// TwinCAT 3 PLC project PLC
// ProgramVersion: 3.1.4024.0
// libraries:
//   Tc2_Standard, * (Beckhoff Automation GmbH)
//   Tc2_System, * (Beckhoff Automation GmbH)
//   Tc3_Module, * (Beckhoff Automation GmbH)
// project tree:
//   / GlobalTextList.TcGTLO, PlcTask.TcTTO, Visualization Manager.TcVMO (not stored), Visualization.TcVIS
//   POUs/ MAIN.TcPOU
// real-time tasks:
//   TASK PlcTask: cycle T#10ms, priority 20, ADS port 350

CONFIGURATION PLC
    RESOURCE PLC ON TwinCAT3
        TASK PlcTask(INTERVAL := T#10ms, PRIORITY := 20);
        PROGRAM MAIN WITH PlcTask : MAIN;
    END_RESOURCE
END_CONFIGURATION

// ---- POUs/MAIN.TcPOU
PROGRAM MAIN
VAR
	StartPb					:	BOOL;
	StopPB					:	BOOL;
	MotorStart				: 	RS;
	Motor					: 	BOOL;
	ProductCnt				: 	CTU;
	LightBarrierSensor		: 	BOOL;
	ProductCounter			: 	WORD;
	TrayChange				: 	BOOL;
END_VAR
VAR // added by the converter: edge detectors and wires of the graphical bodies
    _w1 : ANY;
END_VAR

MotorStart(SET := StartPb, RESET1 := StopPB); // RS
ProductCnt(CU := Motor AND LightBarrierSensor, RESET := _w1, PV := 5); // CTU
ProductCounter := ProductCnt.CV;
Motor := MotorStart.Q1 AND NOT ProductCnt.Q;
_w1 := TrayChange AND ProductCnt.Q;

END_PROGRAM

// ---- GlobalTextList.TcGTLO
TEXTLIST GlobalTextList
  899 = '%s'
  542 = 'Change Tray'
  722 = 'Light Barrier'
  329 = 'Motor'
  959 = 'Please Change the Tray'
  663 = 'Product amount: \n%s'
  828 = 'Product amount: %s'
  814 = 'RUN'
  239 = 'START'
  872 = 'STOP'
END_TEXTLIST

// ---- Visualization.TcVIS
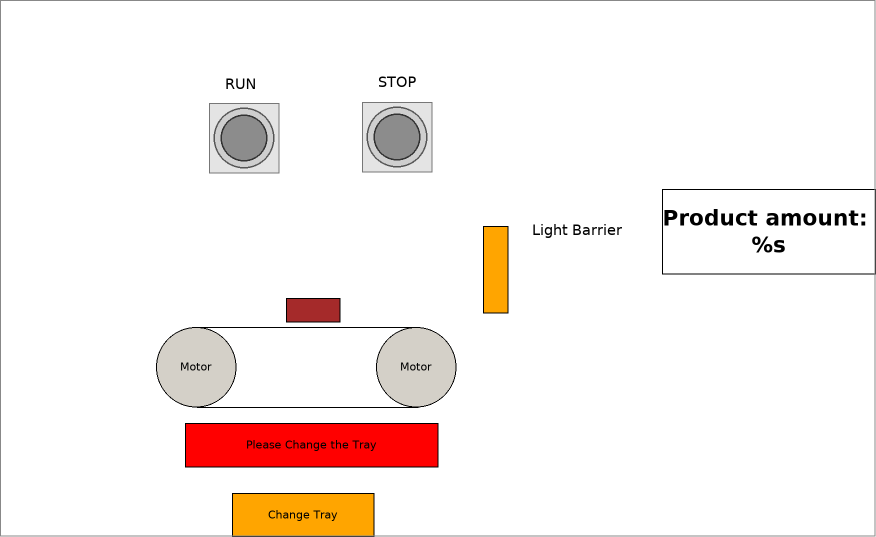
VISUALIZATION Visualization  // 876x537
    PushSwitchLed (209,103 70x70), variable: MAIN.StartPb, behaviour: TAP, style: Switch-PushSwitchLed-Gray
    PushSwitchLed (362,102 70x70), variable: MAIN.StopPB, behaviour: TAP, style: Switch-PushSwitchLed-Gray
    Rectangle (662,189 214x85), "Product amount: %s", text variable: MAIN.ProductCounter
    Ellipse (156,327 80x80), "Motor", colour toggle: MAIN.Motor
    Label (200,69 82x30), "RUN"
    Label (356,67 82x30), "STOP"
    Ellipse (376,327 80x80), "Motor", colour toggle: MAIN.Motor
    Line (197,407) (418,407)
    Line (197,327) (418,327)
    Rectangle (286,298 54x24)
    Rectangle (483,226 25x87), angle 48
        tap MAIN.LightBarrierSensor
    Label (519,215 116x30), "Light Barrier"
    Rectangle (232,493 142x44), "Change Tray", colour toggle: MAIN.ProductCnt.Q
        tap MAIN.TrayChange
    Rectangle (185,423 253x44), "Please Change the Tray", colour toggle: MAIN.ProductCnt.Q, invisible if: NOT MAIN.ProductCnt.Q
END_VISUALIZATION
